Fanuc KAREL source: kt00270.KL

-- PROVISIONAL review KL for V770-1; original PC SHA256 f554d76433d2cc47baad0b778bd75a27f3771c63940b3ffe25906aa34afc6843
-- Incomplete behavior may be omitted. Consult companion uncertainty JSON. Do not deploy.
PROGRAM KT00270
%NOLOCKGROUP
VAR
  OUT : BOOLEAN
-- UNRESOLVED_DECL Y1 type=002018
-- UNRESOLVED_DECL H2 type=002017
BEGIN
  -- UNRESOLVED_PC offsets 5-19; opcodes 2E,22,9D,33,B2
  -- UNRESOLVED_PC offsets 24-38; opcodes 2E,22,9D,33,B4
  -- UNRESOLVED_PC offsets 43-68; opcodes 22,9D,33,B1,22,9D,33,B3,57,23
  -- UNRESOLVED_PC offsets 73-77; opcodes 7F
END KT00270
